(*
    This testsuite runs two tests. One that is enabled (and that is supposed to fail), and one that is disabled (and
    even though it also is failing is not supposed to run).
*)
FUNCTION_BLOCK FB_CreateDisabledTest EXTENDS TcUnit.FB_TestSuite

TestEnabled();
TestDisabled();

METHOD PRIVATE TestDisabled
VAR
    a : BOOL := FALSE;
    b : BOOL := TRUE;
END_VAR
TEST('DISABLED_ThisShouldNotExecute');

AssertEquals(Expected := a,
             Actual := b,
             Message := 'A does not equal B');

TEST_FINISHED();
END_METHOD

METHOD PRIVATE TestEnabled
VAR
    a : BOOL := TRUE;
    b : BOOL := FALSE;
END_VAR
TEST('TestEnabled');

AssertEquals(Expected := a,
             Actual := b,
             Message := 'A does not equal B');

TEST_FINISHED();
END_METHOD

END_FUNCTION_BLOCK

(* stored: Version 1.1.0.1, ProductVersion 3.1.4022.18
   POU FB_CreateDisabledTest: Id {3f1093ff-32d2-455a-8cf0-190014c55a4c}, SpecialFunc None
   Method TestDisabled: Id {773db475-8255-416d-8669-8526d3357b4d}
   Method TestEnabled: Id {aaa74956-ecdb-40ff-a4da-e0ad237c9503} *)
